// TIA Portal V17 export
// export: Created 2024-08-09T12:53:12.0031473Z, ExportSetting WithDefaults, DisplayName Totally Integrated Automation Portal, DisplayVersion V17 Update 7, DisplayName TIA Portal Openness, DisplayVersion V17 Update 7, DisplayName TIA Portal Version Control Interface, DisplayVersion V17, DisplayName STEP 7 Professional, DisplayVersion V17 Update 7, DisplayName STEP 7 Safety, DisplayVersion V17 Update 6, DisplayName WinCC Professional, DisplayVersion V17 Update 7
VAR_GLOBAL   // PLC tag table "Numeros_Circuits"
END_VAR
VAR_GLOBAL CONSTANT   // user constants
   Num_Cir_Exp1 : USInt := 10;
   Num_Cir_Trans_BB01 : USInt := 1;
   Num_Cir_Trans_BB02 : USInt := 2;
   Num_Cir_Trans_TMEL : USInt := 3;
   Num_Cir_Trans_BP1 : USInt := 5;
   Num_Cir_Trans_TMEL2 : USInt := 4;
END_VAR
